METHOD PRIVATE instantiateVoltageOutputs
VAR_INPUT
END_VAR
(*io_module.instantiateVOUT(			
	outPointer:= ADR(sysIO.voltageOutput.coolerPumpDrive_p161),
	byChannel:= lib500_types.IO_VOUT_CHANNEL.IO_VOUT_00
);
*)
io_module.instantiateVOUT(			
	outPointer:= ADR(sysIO.voltageOutput.etsAI5V_p161),
	byChannel:= lib500_types.IO_VOUT_CHANNEL.IO_VOUT_00
);
io_module.instantiateVOUT(			
	outPointer:= ADR(sysIO.voltageOutput.etsAI10V_p185),
	byChannel:= lib500_types.IO_VOUT_CHANNEL.IO_VOUT_01
);
END_METHOD

METHOD PRIVATE instantiatePWDInputs
VAR_INPUT
END_VAR
(*
io_module.instantiatePWD(			
	outPointer:= ADR(sysIO.pwdInput.speedSensor_p115),
	byChannel:= lib500_types.IO_PWD_CHANNEL.IO_PWD_00,
	pwdMode:= lib500_types.IO_PWD_INC_MODE.IO_PWD_INC_2_COUNT,
	byPullType:= lib500_types.IO_PWD_PUPD.IO_PWD_PU_10K,
	readMode:= pwdReadMode.complex,
	wCountInit:= 32767
);
sysIO.pwdInput.speedSensor_p115.pulseMode:= lib500_types.IO_PWD_PULSE_MODE.IO_PWD_HIGH_TIME;
sysIO.pwdInput.speedSensor_p115.freqMode:= lib500_types.IO_PWD_FREQ_MODE.IO_PWD_FALLING_VAR;
*)
END_METHOD

METHOD PRIVATE instantiatePowerStages
VAR_INPUT
END_VAR
io_module.instantiatePower(			
	outPointer:= ADR(sysIO.powerStage.safetySwitch0),
	byChannel:= lib500_types.IO_POWER_CHANNEL.IO_INT_SAFETY_SW_0,
	mode:= lib500_types.IO_POWER_STATE.IO_POWER_ON
);
														
io_module.instantiatePower(			
	outPointer:= ADR(sysIO.powerStage.safetySwitch1),
	byChannel:= lib500_types.IO_POWER_CHANNEL.IO_INT_SAFETY_SW_1,
	mode:= lib500_types.IO_POWER_STATE.IO_POWER_ON
);
														
io_module.instantiatePower(			
	outPointer:= ADR(sysIO.powerStage.safetySwitch2),
	byChannel:= lib500_types.IO_POWER_CHANNEL.IO_INT_SAFETY_SW_2,
	mode:= lib500_types.IO_POWER_STATE.IO_POWER_ON
);
sysIO.powerStage.safetySwitch2.byMinTTCModel:= TTC_580;

														
io_module.instantiatePower(				
	outPointer:= ADR(sysIO.powerStage.powerStage),
	byChannel:= lib500_types.IO_POWER_CHANNEL.IO_INT_POWERSTAGE_ENABLE,
	mode:= lib500_types.IO_POWER_STATE.IO_POWER_ON
);
														
io_module.instantiatePower(			
	outPointer:= ADR(sysIO.powerStage.sensorSupply0),
	byChannel:= lib500_types.IO_POWER_CHANNEL.IO_SENSOR_SUPPLY_0,
	mode:= lib500_types.IO_POWER_STATE.IO_POWER_ON
);
														
io_module.instantiatePower(			
	outPointer:= ADR(sysIO.powerStage.sensorSupply1),
	byChannel:= lib500_types.IO_POWER_CHANNEL.IO_SENSOR_SUPPLY_1,
	mode:= lib500_types.IO_POWER_STATE.IO_POWER_ON
);
														
io_module.instantiatePower(			
	outPointer:= ADR(sysIO.powerStage.sensorSupply2),
	byChannel:= lib500_types.IO_POWER_CHANNEL.IO_SENSOR_SUPPLY_2,
	mode:= lib500_types.IO_POWER_STATE.IO_POWER_ON_10V
);
END_METHOD

METHOD PRIVATE instantiatePWMOutputs
END_METHOD

METHOD PRIVATE instantiateDigitalInputs
VAR_INPUT
END_VAR
END_METHOD

END_PROGRAM

// Device/Application/Modules/IOs/Functions/io_module
PROGRAM io_module
VAR CONSTANT
	DI_maxIndex: 	INT:= 72;
	ADC_maxIndex: 	INT:= 60;
	DO_maxIndex: 	INT:= 40;
	Power_maxIndex: INT:= 10;
	PWM_maxIndex: 	INT:= 36;
	PWD_maxIndex: 	INT:= 19;
	PVG_maxIndex: 	INT:= 7;
	VOUT_maxIndex: 	INT:= 7;
END_VAR
VAR 
	paAllDigitalInputs:  ARRAY[0..DI_maxIndex] 		OF POINTER TO pinDIO;
	paAllADCInputs: 	 ARRAY[0..ADC_maxIndex] 	OF POINTER TO pinADC;		
	paAllDigitalOutputs: ARRAY[0..DO_maxIndex] 		OF POINTER TO pinDIO;
	paAllPowerOutputs: 	 ARRAY[0..Power_maxIndex] 	OF POINTER TO pinPower;
	paAllPWMOutputs:	 ARRAY[0..PWM_maxIndex] 	OF POINTER TO pinPWM;
	paAllPWDInputs:		 ARRAY[0..PWD_maxIndex]		OF POINTER TO pinPWD;
	paAllPVGOutputs:	 ARRAY[0..PVG_maxIndex] 	OF POINTER TO pinPVG;
	paAllVOUTOutputs:	 ARRAY[0..VOUT_maxIndex] 	OF POINTER TO pinVOUT;
	
	iAllDICursor: 	 INT:= 0;
	iAllADCCursor: 	 INT:= 0;	
	iAllDOCursor: 	 INT:= 0;
	iAllPowerCursor: INT:= 0;
	iAllPWMCursor: 	 INT:= 0;
	iAllPWDCursor: 	 INT:= 0;
	iAllPVGCursor: 	 INT:= 0;
	iAllVOUTCursor:	 INT:= 0;
	
	inputPinError: lib500_types.IO_ERRORTYPE;
	outputPinError: lib500_types.IO_ERRORTYPE;
	initializePinError: lib500_types.IO_ERRORTYPE;
	
	byTTCModel: BYTE:= 0;
END_VAR

METHOD PUBLIC instantiateDI: BOOL;
VAR_INPUT
	outPointer: POINTER TO pinDIO;
	byChannel: BYTE;
	byPullType: BYTE:= 0;
END_VAR
instantiateDIO(outPointer, byChannel, byPullType);

paAllDigitalInputs[iAllDICursor]:= outPointer;
iAllDICursor:= iAllDICursor + 1;

IF iAllDICursor >= DI_maxIndex THEN
	iAllDICursor:= 0;
END_IF
END_METHOD

METHOD PUBLIC instantiatePWM
VAR_INPUT
	outPointer: POINTER TO pinPWM;
	byChannel: BYTE;
	wFrequency: WORD;
	bPolarity: BOOL;
	bDiagMargin: BOOL;
END_VAR
outPointer^.byChannel:= byChannel;
outPointer^.wFrequency:= wFrequency;
outPointer^.bPolarity:= bPolarity;
outPointer^.bDiagMargin:= bDiagMargin;

paAllPWMOutputs[iAllPWMCursor]:= outPointer;
iAllPWMCursor:= iAllPWMCursor + 1;

IF iAllPWMCursor >= PWM_maxIndex THEN
	iAllPWMCursor:= 0;
END_IF
END_METHOD

METHOD PUBLIC instantiatePower
VAR_INPUT
	outPointer: POINTER TO pinPower;
	byChannel: BYTE;
	mode: lib500_types.IO_POWER_STATE;
END_VAR
VAR
	pin: pinPower;
END_VAR
outPointer^.byChannel:= byChannel;
outPointer^.mode:= mode;

paAllPowerOutputs[iAllPowerCursor]:= outPointer;
iAllPowerCursor:= iAllPowerCursor + 1;

IF iAllPowerCursor >= Power_maxIndex THEN
	iAllPowerCursor:= 0;
END_IF
END_METHOD

METHOD PUBLIC instantiateVOUT
VAR_INPUT
	outPointer: POINTER TO pinVOUT;
	byChannel: BYTE;
END_VAR
outPointer^.byChannel:= byChannel;

paAllVOUTOutputs[iAllVOUTCursor]:= outPointer;
iAllVOUTCursor:= iAllVOUTCursor + 1;

IF iAllVOUTCursor >= VOUT_maxIndex THEN
	iAllVOUTCursor:= 0;
END_IF
END_METHOD

METHOD PUBLIC instantiateADC
VAR_INPUT
	outPointer: POINTER TO pinADC;
	byChannel: BYTE;
	byPullType: BYTE;
	stADCType: lib500_types.IO_ADC_TYPE;
	stADCRange: lib500_types.IO_ADC_RANGE;
	stADCSensorSupply: lib500_types.IO_SENSOR_SUPPLY;
END_VAR
outPointer^.byChannel:= byChannel;
outPointer^.byPullType:= byPullType;
outPointer^.stADCType:= stADCType;
outPointer^.stADCRange:= stADCRange;
outPointer^.stADCSensorSupply:= stADCSensorSupply;

paAllADCInputs[iAllADCCursor]:= outPointer;
iAllADCCursor:= iAllADCCursor + 1;

IF iAllADCCursor >= ADC_maxIndex THEN
	iAllADCCursor:= 0;
END_IF
END_METHOD

METHOD getInputs : BOOL
VAR
	iDIIterator: INT;
	iADCIterator: INT;
	iPWDIterator: INT;
	pinDITemp: pinDIO;
	pinADCTemp: pinADC;
	pinPWDTemp: pinPWD;
END_VAR
getInputs:= TRUE;
inputPinError:= lib500_types.IO_ERRORTYPE.IO_E_OK;

FOR iDIIterator:= 0 TO iAllDICursor - 1 BY 1 DO
	IF paAllDigitalInputs[iDIIterator] = 0 THEN CONTINUE; END_IF
	IF NOT paAllDigitalInputs[iDIIterator]^.bInitialized THEN CONTINUE; END_IF
	
	pinDITemp:= paAllDigitalInputs[iDIIterator]^;
	IF pinDITemp.byMinTTCModel > byTTCModel THEN CONTINUE; END_IF
	pinDITemp.stError:= lib500.IO_DI_Get(di_channel:= pinDITemp.byChannel, di_value:= ADR(pinDITemp.bValue));	
	
	(* if pin is a negative input negates bValue so that user code can read TRUE if input is active*)
	IF (pinDITemp.byPullType = lib500_types.IO_DI_PUPD.IO_DI_PU_10K) THEN
		pinDITemp.bValue:= NOT(pinDITemp.bValue);
	END_IF
	
	IF (pinDITemp.stError <> lib500_types.IO_ERRORTYPE.IO_E_OK) THEN
		pinDITemp.bValue:= FALSE;
		getInputs:= FALSE;
		inputPinError:= pinDITemp.stError;
	END_IF
	
	paAllDigitalInputs[iDIIterator]^:= pinDITemp;
	
END_FOR



FOR iADCIterator:= 0 TO iAllADCCursor - 1 BY 1 DO
	IF paAllADCInputs[iADCIterator] = 0 THEN CONTINUE; END_IF
	IF NOT paAllADCInputs[iADCIterator]^.bInitialized THEN CONTINUE; END_IF
	
	pinADCTemp:= paAllADCInputs[iADCIterator]^;
	IF pinADCTemp.byMinTTCModel > byTTCModel THEN CONTINUE; END_IF
	pinADCTemp.stError:= lib500.IO_ADC_Get(adc_channel:= pinADCTemp.byChannel, 
											adc_value:= ADR(pinADCTemp.dwValue), 
											fresh:= ADR(pinADCTemp.bValueFresh));
											
	IF pinADCTemp.stError = lib500_types.IO_ERRORTYPE.IO_E_FET_PROT_REENABLE THEN
		lib500.IO_ADC_ResetProtection(adc_channel:= pinADCTemp.byChannel, ADR(pinADCTemp.byResetCount));
	END_IF
	
	IF (pinADCTemp.stError <> lib500_types.IO_ERRORTYPE.IO_E_OK) THEN
		getInputs:= FALSE;
		inputPinError:= pinADCTemp.stError;
	END_IF
	
	paAllADCInputs[iADCIterator]^:= pinADCTemp;
	
END_FOR



FOR iPWDIterator:= 0 TO iAllPWDCursor - 1 BY 1 DO
	IF paAllPWDInputs[iPWDIterator] = 0 THEN CONTINUE; END_IF
	IF NOT paAllPWDInputs[iPWDIterator]^.bInitialized THEN CONTINUE; END_IF
	
	pinPWDTemp:= paAllPWDInputs[iPWDIterator]^;
	IF pinPWDTemp.byMinTTCModel > byTTCModel THEN CONTINUE; END_IF
	pinPWDTemp.stGetVoltageError:= lib500.IO_PWD_GetVoltage(
		pwd_channel:= pinPWDTemp.byChannel,
		voltage:= ADR(pinPWDTemp.uiVoltage),
		fresh:= ADR(pinPWDTemp.bVoltageFresh)
	);
	
	IF pinPWDTemp.bSetIncrementCount THEN
		pinPWDTemp.bSetIncrementCount:= FALSE;
		pinPWDTemp.stIncSetError := lib500.IO_PWD_IncSet(pinPWDTemp.byChannel, pinPWDTemp.wCountZero);
	END_IF
	
	IF pinPWDTemp.readMode = pwdReadMode.incremental THEN 
		pinPWDTemp.stError:= lib500.IO_PWD_IncGet(
								pinPWDTemp.byChannel,
								ADR(pinPWDTemp.wCount),
								ADR(pinPWDTemp.bChannelA),
								ADR(pinPWDTemp.bChannelB)
							);
							
	ELSIF pinPWDTemp.readMode = pwdReadMode.complex THEN 
		pinPWDTemp.stError:= lib500.IO_PWD_ComplexGet(
								timer_channel:= pinPWDTemp.byChannel,
								frequency:= ADR(pinPWDTemp.dwFrequencyHz),
								pulse_width:= ADR(pinPWDTemp.dwPulseWidth),
								pin_value:= ADR(pinPWDTemp.bChannelA),
								pulse_samples:= ADR(pinPWDTemp.pulseSamples)
							);
							
	END_IF	
											
	IF pinPWDTemp.stError = lib500_types.IO_ERRORTYPE.IO_E_FET_PROT_REENABLE THEN
		lib500.IO_PWD_ResetProtection(pwd_channel:= pinPWDTemp.byChannel, ADR(pinPWDTemp.byResetCount));
	END_IF
	
	IF (pinPWDTemp.stError <> lib500_types.IO_ERRORTYPE.IO_E_OK) THEN
		getInputs:= FALSE;
		inputPinError:= pinPWDTemp.stError;
	END_IF
	
	paAllPWDInputs[iPWDIterator]^:= pinPWDTemp;
	
END_FOR
END_METHOD

METHOD PUBLIC instantiatePWD
VAR_INPUT
	outPointer: POINTER TO pinPWD;
	byChannel: BYTE;
	pwdMode: lib500_types.IO_PWD_INC_MODE;
	wCountInit: WORD;
	byPullType: BYTE:= 0;
	readMode: pwdReadMode;
END_VAR
outPointer^.byChannel:= byChannel;
outPointer^.pwdMode:= pwdMode;
outPointer^.wCountInit:= wCountInit;
outPointer^.byPullType:= byPullType;
outPointer^.readMode:= readMode;

paAllPWDInputs[iAllPWDCursor]:= outPointer;
iAllPWDCursor:= iAllPWDCursor + 1;

IF iAllPWDCursor >= PWD_maxIndex THEN
	iAllPWDCursor:= 0;
END_IF
END_METHOD

METHOD PUBLIC initializeIO: BOOL
VAR_INPUT
	TTCModel: BYTE;
END_VAR
VAR
	iDIIterator: INT;
	iDIOterator: INT;
	iADCIterator: INT;
	iPowerChannelIterator: INT;
	iPWMIterator: INT;
	iPWDIterator: INT;
	iPVGIterator: INT;
	iVOUTIterator: INT;
	
	pinDITemp: pinDIO;
	pinDOTemp: pinDIO;
	pinADCTemp: pinADC;
	pinPCTemp: pinPower;
	pinPWMTemp: pinPWM;
	pinPWDTemp: pinPWD;
	pinPVGTemp: pinPVG;
	pinVOUTTemp: pinVOUT;
END_VAR
initializeIO:= TRUE;
initializePinError:= lib500_types.IO_ERRORTYPE.IO_E_OK;
byTTCModel:= TTCModel;


FOR iPowerChannelIterator:= 0 TO iAllPowerCursor - 1 BY 1 DO
	IF paAllPowerOutputs[iPowerChannelIterator] = 0 THEN CONTINUE; END_IF
	pinPCTemp:= paAllPowerOutputs[iPowerChannelIterator]^;
	IF pinPCTemp.bInitialized OR pinPCTemp.byMinTTCModel > byTTCModel THEN CONTINUE; END_IF
	
	pinPCTemp.stInitError:= lib500.IO_POWER_Set(pin:= pinPCTemp.byChannel, mode:= pinPCTemp.mode);										
	pinPCTemp.bInitialized:= (pinPCTemp.stInitError = lib500_types.IO_ERRORTYPE.IO_E_OK);
	IF(pinPCTemp.stInitError <> lib500_types.IO_ERRORTYPE.IO_E_OK) THEN initializePinError:= pinPCTemp.stInitError; END_IF
	IF NOT pinPCTemp.bInitialized THEN initializeIO:= FALSE; END_IF
	
	paAllPowerOutputs[iPowerChannelIterator]^:= pinPCTemp;
	
END_FOR

(* Inputs *)
FOR iADCIterator:= 0 TO iAllADCCursor - 1 BY 1 DO
	IF paAllADCInputs[iADCIterator] = 0 THEN CONTINUE; END_IF
	pinADCTemp:= paAllADCInputs[iADCIterator]^;
	IF pinADCTemp.bInitialized OR pinADCTemp.byMinTTCModel > byTTCModel THEN CONTINUE; END_IF
	
	pinADCTemp.stInitError:= lib500.IO_ADC_ChannelInit(adc_channel:= pinADCTemp.byChannel, 
														pupd:= pinADCTemp.byPullType,
														adc_type:= pinADCTemp.stADCType,
														range:= pinADCTemp.stADCRange,
														sensor_supply:= pinADCTemp.stADCSensorSupply,
														safety_conf:= 0);					
	
	// per qualche motivo K15 init da errore, ma poi funziona la lettura comunque...
	IF pinADCTemp.byChannel = lib500_types.IO_ADC_CHANNEL.IO_ADC_K15 AND pinADCTemp.stInitError = lib500_types.IO_ERRORTYPE.IO_E_CHANNEL_BUSY THEN
		pinADCTemp.stInitError:= lib500_types.IO_ERRORTYPE.IO_E_OK;
	END_IF
	
	IF (pinADCTemp.stInitError <> lib500_types.IO_ERRORTYPE.IO_E_OK) THEN initializePinError:= pinADCTemp.stInitError; END_IF				
	pinADCTemp.bInitialized:= (pinADCTemp.stInitError = lib500_types.IO_ERRORTYPE.IO_E_OK);	
	IF NOT pinADCTemp.bInitialized THEN initializeIO:= FALSE; END_IF
	
	paAllADCInputs[iADCIterator]^:= pinADCTemp;
	
END_FOR

FOR iDIIterator:= 0 TO iAllDICursor - 1 BY 1 DO
	IF paAllDigitalInputs[iDIIterator] = 0 THEN CONTINUE; END_IF
	pinDITemp:= paAllDigitalInputs[iDIIterator]^;
	IF pinDITemp.bInitialized OR pinDITemp.byMinTTCModel > byTTCModel THEN CONTINUE; END_IF
	
	pinDITemp.stInitError:= lib500.IO_DI_Init(di_channel:= pinDITemp.byChannel, pupd:= pinDITemp.byPullType, limits:= 0);		
	IF(pinDITemp.stInitError <> lib500_types.IO_ERRORTYPE.IO_E_OK) THEN initializePinError:= pinDITemp.stInitError; END_IF								
	pinDITemp.bInitialized:= (pinDITemp.stInitError = lib500_types.IO_ERRORTYPE.IO_E_OK);		
	IF NOT pinDITemp.bInitialized THEN	initializeIO:= FALSE; END_IF
	
	paAllDigitalInputs[iDIIterator]^:= pinDITemp;
	
END_FOR




(* Outputs *)

// FOR iDIOterator:= 0 TO iAllDOCursor - 1 BY 1 DO
// 	IF paAllDigitalOutputs[iDIOterator] = 0 THEN CONTINUE; END_IF
// 	pinDOTemp:= paAllDigitalOutputs[iDIOterator]^;
// 	IF pinDOTemp.bInitialized OR pinDOTemp.byMinTTCModel > byTTCModel THEN CONTINUE; END_IF
// 	
// 	pinDOTemp.stInitError:= lib500.IO_DO_Init(do_channel:= pinDOTemp.byChannel, diagnostic:= 0,	safety_conf:= 0);	
// 	IF(pinDOTemp.stInitError <> lib500_types.IO_ERRORTYPE.IO_E_OK) THEN initializePinError:= pinDOTemp.stInitError; END_IF												
// 	pinDOTemp.bInitialized:= (pinDOTemp.stInitError = lib500_types.IO_ERRORTYPE.IO_E_OK);		
// 	IF NOT pinDOTemp.bInitialized THEN initializeIO:= FALSE; END_IF
// 	
// 	paAllDigitalOutputs[iDIOterator]^:= pinDOTemp;
// 	
// END_FOR



FOR iPWMIterator:= 0 TO iAllPWMCursor - 1 BY 1 DO
	IF paAllPWMOutputs[iPWMIterator] = 0 THEN CONTINUE; END_IF
	pinPWMTemp:= paAllPWMOutputs[iPWMIterator]^;
	IF pinPWMTemp.bInitialized OR pinPWMTemp.byMinTTCModel > byTTCModel THEN CONTINUE; END_IF
	
	pinPWMTemp.stInitError:= lib500.IO_PWM_Init(pwm_channel:= pinPWMTemp.byChannel, 
													frequency:= pinPWMTemp.wFrequency,
													polarity:= pinPWMTemp.bPolarity,
													diag_margin:= pinPWMTemp.bDiagMargin,
													safety_conf:= 0);		
								
	IF(pinPWMTemp.stInitError <> lib500_types.IO_ERRORTYPE.IO_E_OK) THEN initializePinError:= pinPWMTemp.stInitError; END_IF		
	pinPWMTemp.bInitialized:= (pinPWMTemp.stInitError = lib500_types.IO_ERRORTYPE.IO_E_OK);		
	IF NOT pinPWMTemp.bInitialized THEN initializeIO:= FALSE; END_IF
	
	paAllPWMOutputs[iPWMIterator]^:= pinPWMTemp;
	
END_FOR



FOR iPWDIterator:= 0 TO iAllPWDCursor - 1 BY 1 DO
	IF paAllPWDInputs[iPWDIterator] = 0 THEN CONTINUE; END_IF
	pinPWDTemp:= paAllPWDInputs[iPWDIterator]^;
	IF pinPWDTemp.bInitialized OR pinPWDTemp.byMinTTCModel > byTTCModel THEN CONTINUE; END_IF
	
	IF pinPWDTemp.readMode = pwdReadMode.incremental THEN
		pinPWDTemp.stInitError:= lib500.IO_PWD_IncInit(
												inc_channel:= pinPWDTemp.byChannel,
												mode:= pinPWDTemp.pwdMode,
												pupd:= pinPWDTemp.byPullType,
												count_init:= pinPWDTemp.wCountInit,
												safety_conf:= 0
								);	
								
	ELSIF pinPWDTemp.readMode = pwdReadMode.complex THEN	
		pinPWDTemp.stInitError:= lib500.IO_PWD_ComplexInit(
			timer_channel:= pinPWDTemp.byChannel, 
			pulse_mode:= pinPwdTemp.pulseMode, 
			freq_mode:= pinPWDTemp.freqMode, 
			capture_count:= pinPWDTemp.byCaptureCount, 
			pupd:= pinPWDTemp.byPullType, 
			safety_conf:= 0
		);
	
	END_IF
								
	IF(pinPWDTemp.stInitError <> lib500_types.IO_ERRORTYPE.IO_E_OK) THEN initializePinError:= pinPWDTemp.stInitError; END_IF	
	pinPWDTemp.bInitialized:= (pinPWDTemp.stInitError = lib500_types.IO_ERRORTYPE.IO_E_OK);		
	IF NOT pinPWDTemp.bInitialized THEN initializeIO:= FALSE; END_IF
	
	paAllPWDInputs[iPWDIterator]^:= pinPWDTemp;

END_FOR



FOR iPVGIterator:= 0 TO iAllPWDCursor - 1 BY 1 DO
	IF paAllPVGOutputs[iPVGIterator] = 0 THEN CONTINUE; END_IF
	pinPVGTemp:= paAllPVGOutputs[iPVGIterator]^;
	IF pinPVGTemp.bInitialized OR pinPVGTemp.byMinTTCModel > byTTCModel THEN CONTINUE; END_IF

	pinPVGTemp.stInitError:= lib500.IO_PVG_Init(pvg_channel:= pinPVGTemp.byChannel, output_value:= pinPVGTemp.wValue);
								
	IF(pinPVGTemp.stInitError <> lib500_types.IO_ERRORTYPE.IO_E_OK) THEN initializePinError:= pinPVGTemp.stInitError; END_IF	
	pinPVGTemp.bInitialized:= (pinPVGTemp.stInitError = lib500_types.IO_ERRORTYPE.IO_E_OK);		
	IF NOT pinPVGTemp.bInitialized THEN initializeIO:= FALSE; END_IF

	paAllPVGOutputs[iPVGIterator]^:= pinPVGTemp;

END_FOR



FOR iVOUTIterator:= 0 TO iAllVOUTCursor - 1 BY 1 DO
	IF paAllVOUTOutputs[iVOUTIterator] = 0 THEN CONTINUE; END_IF
	pinVOUTTemp:= paAllVOUTOutputs[iVOUTIterator]^;
	IF pinVOUTTemp.bInitialized OR pinVOUTTemp.byMinTTCModel > byTTCModel THEN CONTINUE; END_IF
	
	pinVOUTTemp.stInitError:= lib500.IO_VOUT_Init(vout_channel:= pinVOUTTemp.byChannel);	
								
	IF(pinVOUTTemp.stInitError <> lib500_types.IO_ERRORTYPE.IO_E_OK) THEN initializePinError:= pinVOUTTemp.stInitError; END_IF	
	pinVOUTTemp.bInitialized:= (pinVOUTTemp.stInitError = lib500_types.IO_ERRORTYPE.IO_E_OK);		
	IF NOT pinVOUTTemp.bInitialized THEN initializeIO:= FALSE; END_IF
	
	paAllVOUTOutputs[iVOUTIterator]^:= pinVOUTTemp;

END_FOR
END_METHOD

METHOD PUBLIC instantiateDO
VAR_INPUT
	outPointer: POINTER TO pinDIO;
	byChannel: BYTE;
END_VAR
instantiateDIO(outPointer, byChannel, 0);

paAllDigitalOutputs[iAllDOCursor]:= outPointer;
iAllDOCursor:= iAllDOCursor + 1;

IF iAllDOCursor >= DO_maxIndex THEN
	iAllDOCursor:= 0;
END_IF
END_METHOD

METHOD PRIVATE instantiateDIO
VAR_INPUT
	outPointer: POINTER TO pinDIO;
	byChannel: BYTE;
	byPullType: BYTE:= 0;
END_VAR
outPointer^.byChannel:= byChannel;
outPointer^.byPullType:= byPullType;
END_METHOD

METHOD PUBLIC instantiatePVG
VAR_INPUT
	outPointer: POINTER TO pinPVG;
	byChannel: BYTE;
	wValue: WORD:= 5000;
END_VAR
outPointer^.byChannel:= byChannel;
outPointer^.wValue:= wValue;

paAllPVGOutputs[iAllPWDCursor]:= outPointer;
iAllPVGCursor:= iAllPVGCursor + 1;

IF iAllPVGCursor >= PVG_maxIndex THEN
	iAllPVGCursor:= 0;
END_IF
END_METHOD

METHOD setOutputs : BOOL
VAR
	iPowerIterator: INT;
	iDIOterator: INT;
	iPWMIterator: INT;
	iVOUTIterator: INT;
	iPVGIterator: INT;
	
	pinPowerTemp: pinPower;
	pinDOTemp: pinDIO;
	pinPWMTemp: pinPWM;
	pinVOUTTemp: pinVOUT;
	pinPVGTemp: pinPVG;
END_VAR
setOutputs:= TRUE;
outputPinError:= lib500_types.IO_ERRORTYPE.IO_E_OK;

FOR iPowerIterator:= 0 TO iAllPowerCursor - 1 BY 1 DO
	IF paAllPowerOutputs[iPowerIterator] = 0 THEN CONTINUE; END_IF
	pinPowerTemp:= paAllPowerOutputs[iPowerIterator]^;
	IF NOT pinPowerTemp.bInitialized OR pinPowerTemp.byMinTTCModel > byTTCModel THEN CONTINUE; END_IF
	
	pinPowerTemp.stError:= lib500.IO_POWER_Set(
								pin:= pinPowerTemp.byChannel,
								mode:= pinPowerTemp.mode
							);		
		
								
	IF (pinPowerTemp.stError <> lib500_types.IO_ERRORTYPE.IO_E_OK AND pinPowerTemp.stError <> lib500_types.IO_ERRORTYPE.IO_E_NO_DIAG) THEN 
		setOutputs:= FALSE; 
		outputPinError:= pinPowerTemp.stError;
	END_IF		
	
	paAllPowerOutputs[iPowerIterator]^:= pinPowerTemp;	
END_FOR

FOR iDIOterator:= 0 TO iAllDOCursor - 1 BY 1 DO	
	IF paAllDigitalOutputs[iDIOterator] = 0 THEN CONTINUE; END_IF
	pinDOTemp:= paAllDigitalOutputs[iDIOterator]^;
	IF NOT pinDOTemp.bInitialized OR pinDOTemp.byMinTTCModel > byTTCModel THEN CONTINUE; END_IF
	
	pinDOTemp.stError:= lib500.IO_DO_Set(do_channel:= pinDOTemp.byChannel, do_value:= pinDOTemp.bValue);		
													
	pinDOTemp.stErrorGetCut:= lib500.IO_DO_GetCur(do_channel:= pinDOTemp.byChannel, 
													current:= ADR(pinDOTemp.wCurrent),
													fresh:= ADR(pinDOTemp.bCurrentFresh));		
																	
	IF pinDOTemp.stError = lib500_types.IO_ERRORTYPE.IO_E_FET_PROT_REENABLE THEN
		lib500.IO_DO_ResetProtection(do_channel:= pinDOTemp.byChannel, ADR(pinPowerTemp.byResetCount));
	END_IF
	IF pinDOTemp.stError <> lib500_types.IO_ERRORTYPE.IO_E_OK AND pinDOTemp.stError <> lib500_types.IO_ERRORTYPE.IO_E_NO_DIAG AND pinDOTemp.stError <> lib500_types.IO_ERRORTYPE.IO_E_OPEN_LOAD THEN 
		setOutputs:= FALSE; 
		outputPinError:= pinDOTemp.stError;
	END_IF		
	IF pinDOTemp.stErrorGetCut <> lib500_types.IO_ERRORTYPE.IO_E_OK  AND pinDOTemp.stError <> lib500_types.IO_ERRORTYPE.IO_E_NO_DIAG THEN 
		setOutputs:= FALSE; 
		outputPinError:= pinDOTemp.stErrorGetCut;
	END_IF		
							
	paAllDigitalOutputs[iDIOterator]^:= pinDOTemp;	
END_FOR


FOR iPWMIterator:= 0 TO iAllPWMCursor - 1 BY 1 DO
	IF paAllPWMOutputs[iPWMIterator] = 0 THEN CONTINUE; END_IF
	pinPWMTemp:= paAllPWMOutputs[iPWMIterator]^;
	IF NOT pinPWMTemp.bInitialized OR pinPWMTemp.byMinTTCModel > byTTCModel THEN CONTINUE; END_IF
	
	pinPWMTemp.stError:= lib500.IO_PWM_SetDuty(pwm_channel:= pinPWMTemp.byChannel, 
													duty_cycle:= pinPWMTemp.wDuty,
													high_time_fb:= ADR(pinPWMTemp.wFeedbackHighTime),
													period_fb:= ADR(pinPWMTemp.wPeriodFeedback));
													
	pinPWMTemp.stErrorGetCut:= lib500.IO_PWM_GetCur(pwm_channel:= pinPWMTemp.byChannel, 
													current:= ADR(pinPWMTemp.wCurrent),
													fresh:= ADR(pinPWMTemp.bCurrentFresh));		
		
	IF pinPWMTemp.stError = lib500_types.IO_ERRORTYPE.IO_E_FET_PROT_REENABLE THEN
		lib500.IO_PWM_ResetProtection(pwm_channel:= pinPWMTemp.byChannel, ADR(pinPowerTemp.byResetCount));
	END_IF
	
	IF (pinPWMTemp.stError <> lib500_types.IO_ERRORTYPE.IO_E_OK AND pinPWMTemp.stError <> lib500_types.IO_ERRORTYPE.IO_E_NO_DIAG) THEN
		setOutputs:= FALSE; 
		outputPinError:= pinPWMTemp.stError;
	END_IF
	IF pinPWMTemp.stErrorGetCut <> lib500_types.IO_ERRORTYPE.IO_E_OK AND pinPWMTemp.stError <> lib500_types.IO_ERRORTYPE.IO_E_NO_DIAG THEN 
		setOutputs:= FALSE; 
		outputPinError:= pinPWMTemp.stErrorGetCut;
	END_IF		
	
	paAllPWMOutputs[iPWMIterator]^:= pinPWMTemp;	
END_FOR


FOR iVOUTIterator:= 0 TO iAllVOUTCursor - 1 BY 1 DO
	IF paAllVOUTOutputs[iVOUTIterator] = 0 THEN CONTINUE; END_IF
	pinVOUTTemp:= paAllVOUTOutputs[iVOUTIterator]^;
	IF NOT pinVOUTTemp.bInitialized OR pinVOUTTemp.byMinTTCModel > byTTCModel THEN CONTINUE; END_IF
	
	pinVOUTTemp.stError:= lib500.IO_VOUT_SetVoltage(
								vout_channel:= pinVOUTTemp.byChannel,
								output_voltage:= pinVOUTTemp.wOutputVoltageMv
							);		
		
	IF (pinVOUTTemp.stError <> lib500_types.IO_ERRORTYPE.IO_E_OK AND pinVOUTTemp.stError <> lib500_types.IO_ERRORTYPE.IO_E_NO_DIAG) THEN 
		setOutputs:= FALSE; 
		outputPinError:= pinVOUTTemp.stError;
	END_IF		
	
	paAllVOUTOutputs[iVOUTIterator]^:= pinVOUTTemp;	
END_FOR


FOR iPVGIterator:= 0 TO iAllPVGCursor - 1 BY 1 DO
	IF paAllPVGOutputs[iPVGIterator] = 0 THEN CONTINUE; END_IF
	pinPVGTemp:= paAllPVGOutputs[iPVGIterator]^;
	IF NOT pinPVGTemp.bInitialized OR pinPVGTemp.byMinTTCModel > byTTCModel THEN CONTINUE; END_IF
	
	pinPVGTemp.stError:= lib500.IO_PVG_SetOutput(
								pvg_channel:= pinPVGTemp.byChannel,
								output_value:= pinPVGTemp.wValue
							);		
							
	pinPVGTemp.stGetVoltageError := lib500.IO_PVG_GetVoltage(
								pvg_channel:= pinPVGTemp.byChannel,
								voltage:= ADR(pinPVGTemp.uiReadVoltage),
								fresh:= ADR(pinPVGTemp.bVoltageFresh)
							);		
		
	IF pinPVGTemp.stError = lib500_types.IO_ERRORTYPE.IO_E_FET_PROT_REENABLE THEN
		lib500.IO_PVG_ResetProtection(pvg_channel:= pinPVGTemp.byChannel, ADR(pinPowerTemp.byResetCount));
	END_IF
		
	IF (pinPVGTemp.stError <> lib500_types.IO_ERRORTYPE.IO_E_OK AND pinPVGTemp.stError <> lib500_types.IO_ERRORTYPE.IO_E_NO_DIAG) THEN 
		setOutputs:= FALSE; 
		outputPinError:= pinPVGTemp.stError;
	END_IF		
	IF (pinPVGTemp.stGetVoltageError <> lib500_types.IO_ERRORTYPE.IO_E_OK AND pinPVGTemp.stError <> lib500_types.IO_ERRORTYPE.IO_E_NO_DIAG) THEN 
		setOutputs:= FALSE; 
		outputPinError:= pinPVGTemp.stGetVoltageError;
	END_IF
	
	paAllPVGOutputs[iPVGIterator]^:= pinPVGTemp;	
END_FOR
END_METHOD

METHOD PUBLIC mngErrors
VAR_INPUT
END_VAR
ERR.xInputPins:= (inputPinError <> lib500_types.IO_ERRORTYPE.IO_E_OK );
ERR.xOutputPins:= (outputPinError <> lib500_types.IO_ERRORTYPE.IO_E_OK );
ERR.xInitializePins:= (initializePinError <> lib500_types.IO_ERRORTYPE.IO_E_OK );
END_METHOD

END_PROGRAM

// Device/Application/Modules/J1939/J1939_PRG
PROGRAM J1939_PRG
VAR_INPUT	
	canbus: canBus;
	xInitialized: BOOL:= FALSE;
END_VAR
VAR CONSTANT
	PGN_ONREQ_COUNT: UINT:= 4;
END_VAR
VAR	
	uiLifetimeMs: UINT;
	stJ1939ReceiveMask: canReceiveMask;
	uiPGNRequestSendTimerMs: UINT:= 0;
	byPGNRequestCursor: BYTE:= 0;
	uiaPGNRequestIDs: ARRAY[0..PGN_ONREQ_COUNT-1] OF UINT:= [
		//16#C100,
		16#FEE9,
		16#FEDC,
		//16#FEEB,
		//16#FEDA,
		//16#FEC0,
		16#FEE5,
		16#FDC6
	];
END_VAR

IF NOT xInitialized THEN
	xInitialized:= initReceiveMasks();
ELSE
	receiveMessage();
	IF J1939.xSendPGNRequest THEN sendPGNRequests(); END_IF
END_IF

mngEngineStatus();

Utils.decrementUINT(uiLifetimeMs, 10);

METHOD PRIVATE initReceiveMasks: BOOL;
VAR
	xRet: BOOL:= FALSE;
END_VAR
IF canbus.bActive AND canbus.stChannel.bInitialized THEN
	xRet:= TRUE;
	
	registerReceiveMask(stCanBus:=canbus, udiId:= 16#FFFFFF00, receiveMask:= stJ1939ReceiveMask, udiCobIdMask:= 16#000000FF);
	IF NOT stJ1939ReceiveMask.bInitialized THEN xRet:= FALSE; END_IF

END_IF

initReceiveMasks:= xRet;
END_METHOD

METHOD PRIVATE receiveMessage
VAR CONSTANT
	MAX_RCV_LOOP: UINT:= 100;
END_VAR
VAR
	uiReceivedMsgs: UINT:= 0;
	hMsg: DWORD;
	ctMsgLeft: CL2.CAA.COUNT;
	faulta: CL2.CAA.ERROR;
	udiId: UDINT;
	usiaData: ARRAY[0..7] OF USINT;
END_VAR
REPEAT
	//receive a message from hReceiver
	hMsg := CL2.Read(hReceiverId := stJ1939ReceiveMask.stCAAMask, pctMsgLeft := ADR(ctMsgLeft), peError := ADR(faulta));
	IF hMsg <> 0 THEN
		uiLifetimeMs:= 3000;
		udiId:= CL2.GetMessageId(hMsg, 0);
		usiaData:= CL2.GetMessageDataPointer(hMsg, 0)^;
		
		parseMessage(
			udiMsgId:= udiId, 
			usiData:= usiaData
		);
		
		IF J1939.xRedirectMessages THEN
			redirectToDisplay(
				udiMsgId:= udiId, 
				usiData:= usiaData
			);
		END_IF
		
		CL2.FreeMessage(hMsg); //release message
		hMsg := 0; //to avoid using an already released message
		
	END_IF
UNTIL (ctMsgLeft = 0 OR uiReceivedMsgs > MAX_RCV_LOOP)
END_REPEAT
END_METHOD

METHOD PRIVATE parseMessage
VAR_INPUT	
	udiMsgId: UDINT;
	usiData: ARRAY [0..7] OF USINT;
END_VAR
VAR
	uiPGN: UINT;
	rTmp: REAL;
END_VAR
uiPGN:= UDINT_TO_UINT(SHR(udiMsgId AND 16#00FFFF00, 8));

CASE uiPGN OF
	16#C100:
		J1939.uiMinutesRunWhileMILAct:= Utils.bytesToUInt16(usiData[5], usiData[4]);
		
	16#F004:
		J1939.iTorquePercent:= USINT_TO_INT(usiData[2]) -125;
		J1939.uiEngineSpeedRpm:= REAL_TO_UINT(Utils.bytesToUReal16(usiData[4], usiData[3]) * 0.125);
		
	16#FEE9:
		J1939.lrEngineTotalFuelUsedLiters:= (UDINT_TO_REAL(Utils.bytesToUDInt32(usiData[4], usiData[5], usiData[6], usiData[7])) * 0.5);
		
	16#FEF2:
		J1939.rEngineFuelRateLph:= Utils.bytesToUReal16(usiData[1], usiData[0]) * 0.05;
		
	16#FEF5:
		J1939.byBarometricPressureKPa:= REAL_TO_BYTE(USINT_TO_REAL(usiData[0]) * 0.5);	
		J1939.iAmbientAirTemperatureDegC:= REAL_TO_INT((Utils.bytesToUReal16(usiData[4], usiData[3]) * 0.03125)-273);	
		J1939.iEngineIntakeAirTemperatureDegC:= USINT_TO_INT(usiData[5]) - 40;	
		
	16#FEEF:
		J1939.uiOilPressureKPa:= usiData[3] * 4;	
		J1939.byCoolantLevelPerc:= REAL_TO_BYTE(BYTE_TO_REAL(usiData[7]) * 0.4);	
		
	16#FEEE:
		J1939.iEngineCoolantTempDegC:= USINT_TO_INT(usiData[0]) - 40;	
		J1939.iEngineFuelTempDegC:= USINT_TO_INT(usiData[1]) - 40;	
		
	16#FDB4:
		J1939.iAftertreatmentDPFIntakeGasTempDegC:= (REAL_TO_INT(Utils.bytesToUReal16(usiData[3], usiData[2]) * 0.03125))-273;	
			
	16#FE56:
		;// non chiaro
		
	16#FEF7:
		rTmp:= Utils.bytesToUReal16(usiData[5], usiData[4]);
		IF rTmp = 16#FFFF THEN rTmp:= 0; END_IF
		J1939.rBatteryPotentialV:= rTmp * 0.05;	
		
	16#FDC6:
		J1939.byEngineStartEnable:= usiData[0] AND 16#03;	
		
	16#FEDC:
		J1939.rEngineTotalIdleHours:= (UDINT_TO_REAL(Utils.bytesToUDInt32(usiData[4],usiData[5],usiData[6],usiData[7])) * 0.05);	
		
	16#FC31:
		J1939.byAftertreatmentEngineSpeedIncreaseRequest:= SHR(usiData[0], 4) AND 16#03;	

	16#FEE3:
		;// non chiaro
		
	16#FEEB:
		;// non chiaro

	16#FEE4:
		J1939.byEngineWaitToStartLamp:= usiData[3] AND 16#03;	
		J1939.byEngineIdleShutdownStatus:= usiData[0] AND 16#03;	
		J1939.byEngineIdleShutdownAlert:= SHR(usiData[0], 2) AND 16#03;	
		
	16#FEDA:
		;// non chiaro

	16#FEC0:
		J1939.byServiceComponentId1:= usiData[0];
		J1939.byServiceComponentId2:= usiData[3];
		J1939.byServiceComponentId3:= usiData[5];	
		J1939.iServiceDelayHours:= UINT_TO_INT(Utils.bytesToUInt16(usiData[7],usiData[6])) - 32127;	

	16#FEE5:
		J1939.rEngineTotalOperationHours:= (UDINT_TO_REAL(Utils.bytesToUDInt32(usiData[0],usiData[1],usiData[2],usiData[3])) * 0.05);	
	
	16#FD7C:
		J1939.byDPFFilterLamp:= usiData[0] AND 16#07;	
		J1939.byAftertreatmentDPFActiveRegeneration:= SHR(usiData[1], 2) AND 16#03;	
		J1939.byAftertreatmentDPFFilterStatus:= SHR(usiData[1], 4) AND 16#07;	
		J1939.byDPFActiveRegenerationInhibitedDueSwitch:= SHR(usiData[2], 2) AND 16#03;	
		J1939.byDPFActiveRegenerationInhibitedDueTmpSysLock:= usiData[5] AND 16#03;	
		J1939.byDPFActiveRegenerationInhibitedDuePermSysLock:= SHR(usiData[5], 2) AND 16#03;	
		
	16#FECA:
		J1939.byWarningIndicator:= SHR(usiData[0], 2) AND 16#03;	
		J1939.byWarningIndicatorFlash:= SHR(usiData[1], 2) AND 16#03;
		J1939.byShutdownIndicator:= SHR(usiData[0], 4) AND 16#03;
		J1939.byEngineProtectIndicator:= SHR(usiData[0], 0) AND 16#03;
		J1939.byEngineProtectIndicatorFlash:= SHR(usiData[1], 0) AND 16#03;
		J1939.byEmissionSystemMalfunctionIndicator:= SHR(usiData[0], 6) AND 16#03;
		J1939.byEmissionSystemMalfunctionIndicatorFlash:= SHR(usiData[1], 6) AND 16#03;

		J1939.DM1_SPN:= usiData[2];
		J1939.DM1_SPN:= J1939.DM1_SPN OR SHL(BYTE_TO_ULINT(usiData[3]), 8);
		J1939.DM1_SPN:= J1939.DM1_SPN OR SHL(BYTE_TO_ULINT(usiData[4] AND 16#E0), 16);
		IF J1939.DM1_SPN = 16#7FFFF THEN J1939.DM1_SPN:= 0; END_IF
		J1939.DM1_FMI:= usiData[4] AND 16#1F;
		IF J1939.DM1_FMI = 16#1F THEN J1939.DM1_FMI:= 0; END_IF
		J1939.DM1_OC:= usiData[5] AND 16#7F;
		IF J1939.DM1_OC = 16#7F THEN J1939.DM1_OC:= 0; END_IF
		
	16#FD0C: // NON C'E'
		// J1939.xLowOilPressure:= (SHR(usiData[1], 4) AND 16#03) = 1;	
	
END_CASE
END_METHOD

METHOD PRIVATE sendPGNRequests
VAR
	i: INT;
	msg: canMessage;
END_VAR
Utils.decrementUINT(uiPGNRequestSendTimerMs, 10);
IF uiPGNRequestSendTimerMs > 0 THEN RETURN; END_IF
uiPGNRequestSendTimerMs:= 100;

msg.bExtended:= TRUE;
msg.byLength:= 3;
msg.udiId:= 16#18EAFF00;
msg.udiId:= msg.udiId OR J1939.byECUNodeId;
msg.byaData[0]:= UINT_TO_BYTE(SHR(uiaPGNRequestIDs[byPGNRequestCursor], 0) AND 16#FF);
msg.byaData[1]:= UINT_TO_BYTE(SHR(uiaPGNRequestIDs[byPGNRequestCursor], 8) AND 16#FF);
msg.byaData[2]:= 0;

byPGNRequestCursor:= byPGNRequestCursor+1;
IF byPGNRequestCursor >= PGN_ONREQ_COUNT THEN 
	byPGNRequestCursor:= 0;
END_IF

sendMessage(stCanBus:= canbus, stMessageToSend:= msg);
END_METHOD

METHOD PUBLIC mngEngineStatus
VAR_INPUT
END_VAR
J1939.xEngineOnline:= uiLifetimeMs > 0;

J1939.xEngineRunning:= J1939.xEngineOnline AND (J1939.uiEngineSpeedRpm > 300);
J1939.xEngineDPFRegenActive:= J1939.xEngineOnline AND (J1939.byAftertreatmentDPFActiveRegeneration = 1);
J1939.xEngineDPFRegenRequest:= J1939.xEngineOnline AND (J1939.byAftertreatmentDPFActiveRegeneration = 2);

J1939.xLowOilPressure:= (J1939.uiOilPressureKPa < 90);

J1939.xEngineLamp:= (
		J1939.byWarningIndicator = 1 OR	
		J1939.byWarningIndicatorFlash = 1 OR	
		J1939.byEngineProtectIndicator = 1 OR	
		J1939.byEngineProtectIndicatorFlash = 1 OR	
		J1939.byEmissionSystemMalfunctionIndicator = 1 OR	
		J1939.byEmissionSystemMalfunctionIndicatorFlash = 1
);	

J1939.xEngineLampRed:= (
	J1939.byShutdownIndicator = 1
);
END_METHOD

METHOD PRIVATE redirectToDisplay
VAR_INPUT	
	udiMsgId: UDINT;
	usiData: ARRAY [0..7] OF USINT;
END_VAR
VAR
	msg: canMessage;
	i: INT;
END_VAR
msg.udiId:= udiMsgId;
msg.byLength:= 8;
msg.bExtended:= TRUE;
FOR i:= 0 TO 7 DO
	msg.byaData[i]:= USINT_TO_BYTE(usiData[i]);
END_FOR

sendMessage(stCanBus:= fieldbus.can[2], stMessageToSend:= msg);
END_METHOD

END_PROGRAM

// Device/Application/Program logic/UI_PRG
PROGRAM UI_PRG
VAR
	blinker_100ms: BLINK;
	blinker_500ms: BLINK;
END_VAR

blinker_100ms(ENABLE:= TRUE, TIMELOW:= T#100MS, TIMEHIGH:= T#100MS, OUT=> ui.xBlinker_100ms);
blinker_500ms(ENABLE:= TRUE, TIMELOW:= T#500MS, TIMEHIGH:= T#500MS, OUT=> ui.xBlinker_500ms);

END_PROGRAM

// Device/Application/Program logic/mngCanbusStatus
PROGRAM mngCanbusStatus
VAR
	iCanIterator: INT;
	bTmpCanToReinit: BOOL;
	tmpCanStatus: CanHandleStatus;
	handleCloseError: CL2.ERROR;
END_VAR

FOR iCanIterator:= 0 TO fieldbus.iCanbusCount-1 BY 1 DO	
	IF (fieldbus.can[iCanIterator].stChannel.bInitialized) AND fieldbus.can[iCanIterator].bActive THEN
		
		tmpCanStatus:= checkCanBusStatus(
							hDriver:= fieldbus.can[iCanIterator].stChannel.driver, 
							bDriverToReinitialize=> bTmpCanToReinit
						);
						
		IF bTmpCanToReinit THEN
			handleCloseError:= CL2.DriverClose(hDriver:= fieldbus.can[iCanIterator].stChannel.driver);
			fieldbus.can[iCanIterator].stChannel.driver:= CL2.CAA.gc_hINVALID;
			fieldbus.can[iCanIterator].stChannel.bInitialized:= FALSE;
			
			fieldbus.bCanbusInitialized:= initializeCanbus();
			J1939_PRG.xInitialized:= FALSE; // triggers receive mask recreation
		END_IF
		
	END_IF		
END_FOR

METHOD PUBLIC checkCanBusStatus: CanHandleStatus;
VAR_INPUT
	hDriver: CL2.CAA.HANDLE;
END_VAR

VAR_OUTPUT
	bDriverToReinitialize: BOOL;
END_VAR

VAR
	handlerStatus: CanHandleStatus;
	uidFreeMessagesInPoll: UDINT;
	uidMessagesInElabQueue: UDINT;
END_VAR
uidFreeMessagesInPoll:= CL2.GetReceivePoolSize(hDriver, 0);
uidMessagesInElabQueue:= CL2.GetReceiveQueueLength(hDriver, 0);
IF uidFreeMessagesInPoll < CONST.CANBUS_MIN_FREE_POLL OR uidMessagesInElabQueue > CONST.CANBUS_MAX_RX_QUEUE THEN
	ERR.xCanbusHeavy:= TRUE;
	bDriverToReinitialize:= TRUE;
END_IF

handlerStatus.uidFreeMessagesInPoll:= uidFreeMessagesInPoll;
handlerStatus.uidMessagesInElabQueue:= uidMessagesInElabQueue;

checkCanBusStatus:= handlerStatus;
END_METHOD

END_PROGRAM

// Device/Application/Program logic/initializeCanbus
FUNCTION initializeCanbus : BOOL
VAR_INPUT
END_VAR

VAR
	iCanIterator: INT;
	bTempCanbusInitialized: BOOL:= FALSE;
END_VAR

(* initialization of all canbus channels activated by usercode (bActive flag) *)
FOR iCanIterator:= 0 TO fieldbus.iCanbusCount-1 BY 1 DO	
	IF (NOT fieldbus.can[iCanIterator].stChannel.bInitialized) AND fieldbus.can[iCanIterator].bActive THEN			
		fieldbus.can[iCanIterator].stChannel.usiChannel:= INT_TO_USINT(iCanIterator);
		fieldbus.can[iCanIterator].stChannel.uiBaudrateKbps:= fieldbus.uiaCanBaudrates[iCanIterator];
		initializeCanHandle(stCanBus:=fieldbus.can[iCanIterator]);								
	END_IF		
END_FOR

(* check if all activated channels are correctly initialized *)
bTempCanbusInitialized:= TRUE;	
FOR iCanIterator:= 0 TO fieldbus.iCanbusCount-1 BY 1 DO
	IF(fieldbus.can[iCanIterator].bActive AND (NOT fieldbus.can[iCanIterator].stChannel.bInitialized)) THEN
		bTempCanbusInitialized:= FALSE;
		EXIT;
	END_IF
END_FOR

initializeCanbus:= bTempCanbusInitialized;

END_FUNCTION

// Device/Application/Modules/Canbus/Functions/initializeCanHandle
// This PRG contains non safety-related code.
// The following attribute is autogenerated. Do not remove.
{attribute 'location':='16#800'}
PROGRAM initializeCanHandle
VAR_IN_OUT
	stCanBus: canBus;
END_VAR

IF(stCanBus.stChannel.driver = CL2.CAA.gc_hINVALID) THEN
	stCanBus.stChannel.driver := CL2.DriverOpenH(
		usiNetId := stCanBus.stChannel.usiChannel, 
		uiBaudrate := stCanBus.stChannel.uiBaudrateKbps, 
		xSupport29Bits := TRUE, 
		ctMessages := 50, 
		peError := ADR(stCanBus.stChannel.initializeError)
	);		
	IF stCanBus.stChannel.driver <> CL2.CAA.gc_hINVALID  THEN
		stCanBus.stChannel.bInitialized := TRUE;
	END_IF
END_IF

END_PROGRAM

// Device/Application/Modules/Canbus/Safety interface/Functions/safeSendMessage
PROGRAM safeSendMessage
VAR_IN_OUT
	stCanBus: canBus;
END_VAR
VAR_INPUT
	stMessageToSend: canMessage;
END_VAR
VAR
	iTransMsgPointer: INT:= 0;
END_VAR

FOR iTransMsgPointer:= 0 TO canGVL.iTransmitBufferSize-1 BY 1 DO
	IF(stCanBus.stTransmitBuffer[iTransMsgPointer].udiId = 0) THEN
		stCanBus.stTransmitBuffer[iTransMsgPointer]:= stMessageToSend;
		EXIT;
	END_IF
END_FOR

END_PROGRAM

// Device/Application/Modules/Canbus/Safety interface/Functions/safetyCanbusInterface
PROGRAM safetyCanbusInterface
VAR_INPUT
END_VAR
VAR_OUTPUT
END_VAR
VAR
END_VAR

END_PROGRAM

// Device/Application/Modules/Canbus/Safety interface/Tasks/CAN_PRG_SAFE
PROGRAM CAN_PRG_SAFE
VAR_INPUT
END_VAR
VAR_OUTPUT
END_VAR
VAR
END_VAR

exchangeVariables();

METHOD exchangeVariables
VAR
	iBusCursor: INT;
END_VAR
(* unsafe --> safe *)
IF canEVL.bChannelsHasChanges THEN	
	FOR iBusCursor:= 0 TO canGVL.iBusCount-1 BY 1 DO	
		canGVL.busses[iBusCursor].stChannel:= canGVL.busses[iBusCursor].stChannel;
	END_FOR
	canEVL.bChannelsHasChanges:= FALSE;	
	
ELSIF canEVL.bTransmitBuffersHasChanges THEN	
	FOR iBusCursor:= 0 TO canGVL.iBusCount-1 BY 1 DO	
		canGVL.busses[iBusCursor].stTransmitBuffer:= canGVL.busses[iBusCursor].stTransmitBuffer;
	END_FOR	
	canEVL.bTransmitBuffersHasChanges:= FALSE;
	
ELSIF canEVL.bMasksHasChanges THEN	
	FOR iBusCursor:= 0 TO canGVL.iBusCount-1 BY 1 DO	
		canGVL.busses[iBusCursor].staReceiveMasks:= canGVL.busses[iBusCursor].staReceiveMasks;
	END_FOR	
	canEVL.bMasksHasChanges:= FALSE;
	
END_IF
END_METHOD

END_PROGRAM

// Device/Application/Modules/Canbus/Safety interface/Tasks/CAN_PRG_UNSAFE
// This PRG contains non safety-related code.
// The following attribute is autogenerated. Do not remove.
{attribute 'location':='16#800'}
PROGRAM CAN_PRG_UNSAFE
VAR_INPUT
END_VAR
VAR_OUTPUT
END_VAR
VAR
	iBusCursor: INT:= 0;
	iTransMsgPointer: INT:= 0;
	iReceiveMaskPointer: INT:= 0;
END_VAR

FOR iBusCursor:= 0 TO canGVL.iBusCount-1 BY 1 DO
	
	IF( canGVL.busses[iBusCursor].bActive AND (NOT canGVL.busses[iBusCursor].stChannel.bInitialized) ) THEN
		(* Inizializzazione canali *)
		canEVL.busses[iBusCursor]:= canGVL.busses[iBusCursor];
		initializeCanHandle(stCanBus:=canEVL.busses[iBusCursor]);
		IF canEVL.busses[iBusCursor].stChannel.bInitialized THEN canEVL.bChannelsHasChanges:= TRUE; END_IF;
		
	ELSIF( canGVL.busses[iBusCursor].bActive AND canGVL.busses[iBusCursor].stChannel.bInitialized ) THEN
		
		(* Creazione maschere di ricezione *)
		FOR iReceiveMaskPointer:= 0 TO canGVL.iReceiveMaskCount-1 BY 1 DO
			IF(canGVL.busses[iBusCursor].staReceiveMasks[iReceiveMaskPointer].bActive AND NOT canGVL.busses[iBusCursor].staReceiveMasks[iReceiveMaskPointer].bInitialized) THEN
				registerReceiveMask(stCanBus:= canGVL.busses[iBusCursor], 
									udiId:= canGVL.busses[iBusCursor].staReceiveMasks[iReceiveMaskPointer].udiId,
									receiveMask:= canEVL.busses[iBusCursor].staReceiveMasks[iReceiveMaskPointer]
									); 
				canEVL.bMasksHasChanges:= TRUE;
			END_IF
		END_FOR
		
		(* Invio messaggi *)
		FOR iTransMsgPointer:= 0 TO canGVL.iTransmitBufferSize-1 BY 1 DO
			IF(canGVL.busses[iBusCursor].stTransmitBuffer[iTransMsgPointer].udiId > 0) THEN
				sendMessage(stCanBus:= canGVL.busses[iBusCursor], stMessageToSend:= canGVL.busses[iBusCursor].stTransmitBuffer[iTransMsgPointer]);
				canEVL.busses[iBusCursor].stTransmitBuffer[iTransMsgPointer].udiId:= 0;

				canEVL.bTransmitBuffersHasChanges:= TRUE;
			END_IF
		END_FOR	 
		
	END_IF
	
END_FOR

END_PROGRAM

// Device/Application/Modules/Canbus/Safety interface/Functions/safeRegisterReceiveMask
PROGRAM safeRegisterReceiveMask
VAR_IN_OUT
	stCanBus: canBus;
END_VAR
VAR_INPUT
	udiId: UDINT:= 0;
END_VAR
VAR_OUTPUT
	iMaskCursor: INT:= -1;
END_VAR
VAR
	iReceiveMaskCursor: INT:= 0;
	stNewReceiveMask: canReceiveMask;
END_VAR

FOR iReceiveMaskCursor:= 0 TO canGVL.iReceiveMaskCount-1 BY 1 DO
	IF(NOT stCanBus.staReceiveMasks[iReceiveMaskCursor].bActive) THEN
		stNewReceiveMask.udiId:= udiId;
		stNewReceiveMask.bActive:= TRUE;
		stCanBus.staReceiveMasks[iReceiveMaskCursor]:= stNewReceiveMask;
		iMaskCursor:= iReceiveMaskCursor;
		EXIT;
	END_IF
END_FOR

END_PROGRAM

// Device/Application/Visualization
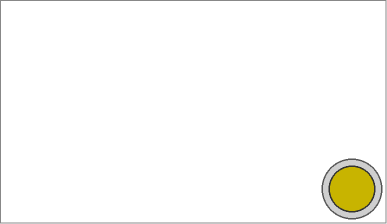
VISUALIZATION Visualization  // 387x224
    Lamp1 (317,154 70x70), invisible if: system.machineModel = 1, style: Lamp-Lamp1-Yellow
END_VISUALIZATION
